(********************* G.D S.p.A. - Technical Department ***********************************
This program has been generated automatically from Application Designer DE&F
********************************************************************************************)
PROGRAM dbg_csp_case_feed_shuttle_sensors
VAR
  part_present_ls_di_shd : digital_input_shadow;
  part_present_os_di_shd : digital_input_shadow;
END_VAR

_objects_manager();

IF	g_application_status <> APPLICATION_STATUS_RUNNING
THEN
	RETURN;
END_IF

CASE process_get_mode(CONVERSION_this := dbg_root.prc) OF
	MODE_ABSENT,
	MODE_INACTIVE:
		RETURN;
	MODE_TEST:
		RETURN;
END_CASE

ACTION _objects_manager:
IF	objects_initialization()
THEN
	digital_input_shadow_init(
		sim_mode:= SHADOW_SIMULATION_MODE_AUTOMATIC, 
		father:= csp_case_feed_shuttle_sensors.part_present_ls_di, 
		process:= dbg_root.prc, 
		CONVERSION_this:= part_present_ls_di_shd);

	digital_input_shadow_init(
		sim_mode:= SHADOW_SIMULATION_MODE_AUTOMATIC, 
		father:= csp_case_feed_shuttle_sensors.part_present_os_di, 
		process:= dbg_root.prc, 
		CONVERSION_this:= part_present_os_di_shd);

	RETURN;
END_IF

IF	objects_running()
THEN
	digital_input_shadow_cycle(part_present_ls_di_shd);
	digital_input_shadow_cycle(part_present_os_di_shd);
END_IF
END_ACTION

END_PROGRAM

(* stored: Version 1.1.0.1, ProductVersion 3.1.4022.12
   POU dbg_csp_case_feed_shuttle_sensors: Id {b8469b28-01bc-4914-bea6-23d36cd46c76}, SpecialFunc None
   Action _objects_manager: Id {a5d7ea93-86b9-41a0-a310-2d9eb4ea2573} *)
